// Mitsubishi GX Works2 project: 멜섹 485 통신 온도계   PLC: Q03UDV

PROGRAM MAIN
VAR
  u2k2k1 : BOOL;
  k2k1 : BOOL;
END_VAR
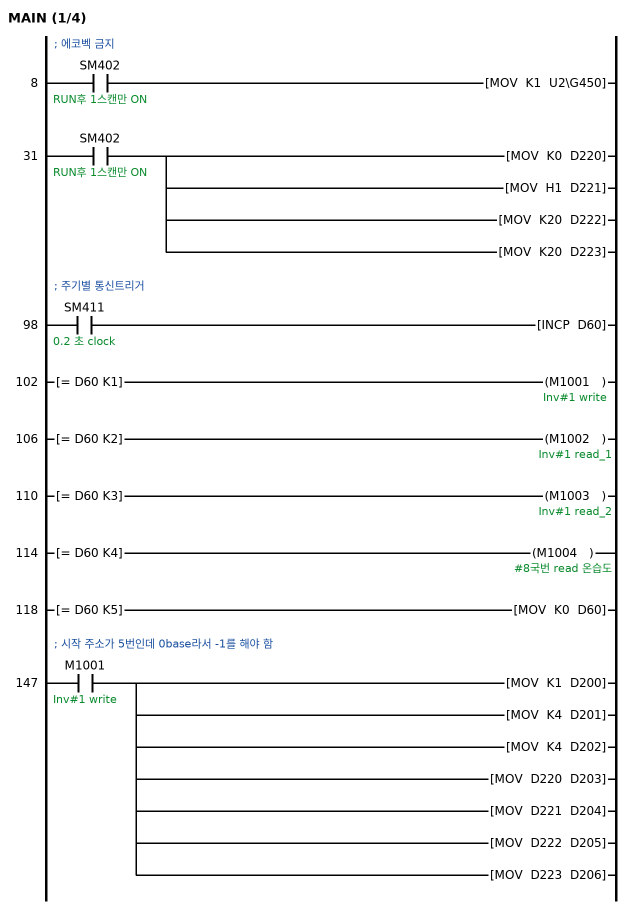
; 에코벡 금지
8     LD      SM402  ; RUN후 1스캔만 ON
      MOV     K1 U2\G450
        [note] 에코벡을 1로 만들어서 금지 시킴
31    LD      SM402  ; RUN후 1스캔만 ON
      MOV     K0 D220
        [note] 인버터 주파수 0hz설정
      MOV     H1 D221
        [note] 인버터 정지 값 1로만듬
      MOV     K20 D222
        [note] 가속 시간 초기값
      MOV     K20 D223
        [note] 감속 시간 초기값
; 주기별 통신트리거
98    LD      SM411  ; 0.2 초 clock
      INCP    D60
102   LD=     D60 K1
      OUT     M1001  ; Inv#1 write
106   LD=     D60 K2
      OUT     M1002  ; Inv#1 read_1
110   LD=     D60 K3
      OUT     M1003  ; Inv#1 read_2
114   LD=     D60 K4
      OUT     M1004  ; #8국번 read 온습도
118   LD=     D60 K5
      MOV     K0 D60
; 시작 주소가 5번인데 0base라서 -1를 해야 함
147   LD      M1001  ; Inv#1 write
      MOV     K1 D200
        [note] ; #1 WRITE DATA PLC>INV설정
      MOV     K4 D201
        [note] 5번인데 0base라서 -1를 한다
      MOV     K4 D202
      MOV     D220 D203
      MOV     D221 D204
      MOV     D222 D205
      MOV     D223 D206
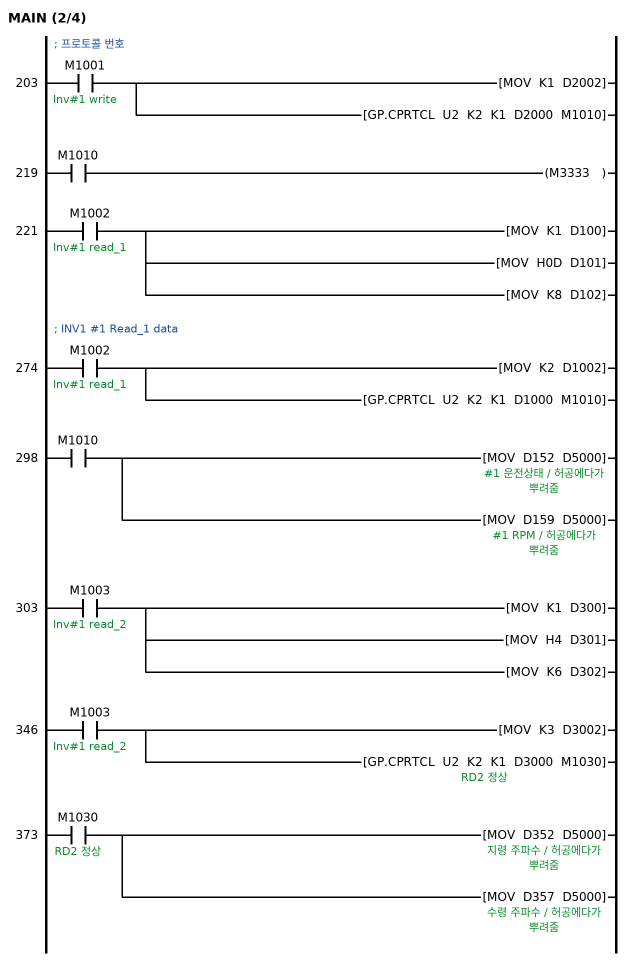
; 프로토콜 번호
203   LD      M1001  ; Inv#1 write
      MOV     K1 D2002
      GP.CPRTCL U2 K2 K1 D2000 M1010
219   LD      M1010
      OUT     M3333
221   LD      M1002  ; Inv#1 read_1
      MOV     K1 D100
        [note] SLAVE ADRESS #1
      MOV     H0D D101
        [note] START ADDRESS 000E-1=H0D
      MOV     K8 D102
        [note] 워드 주소개수
; INV1 #1 Read_1 data
274   LD      M1002  ; Inv#1 read_1
      MOV     K2 D1002
        [note] 프로토콜 2번
      GP.CPRTCL U2 K2 K1 D1000 M1010
298   LD      M1010
      MOV     D152 D5000  ; #1 운전상태 / 허공에다가 뿌려줌
      MOV     D159 D5000  ; #1 RPM
303   LD      M1003  ; Inv#1 read_2
      MOV     K1 D300
        [note] slave address #1
      MOV     H4 D301
        [note] start adress 5 -1
      MOV     K6 D302
        [note] 워드 주소갯수 6개 최대 8개
346   LD      M1003  ; Inv#1 read_2
      MOV     K3 D3002
        [note] 프로토콜 번호 3번
      GP.CPRTCL U2 K2 K1 D3000 M1030  ; RD2 정상
373   LD      M1030  ; RD2 정상
      MOV     D352 D5000  ; 지령 주파수
      MOV     D357 D5000  ; 수령 주파수
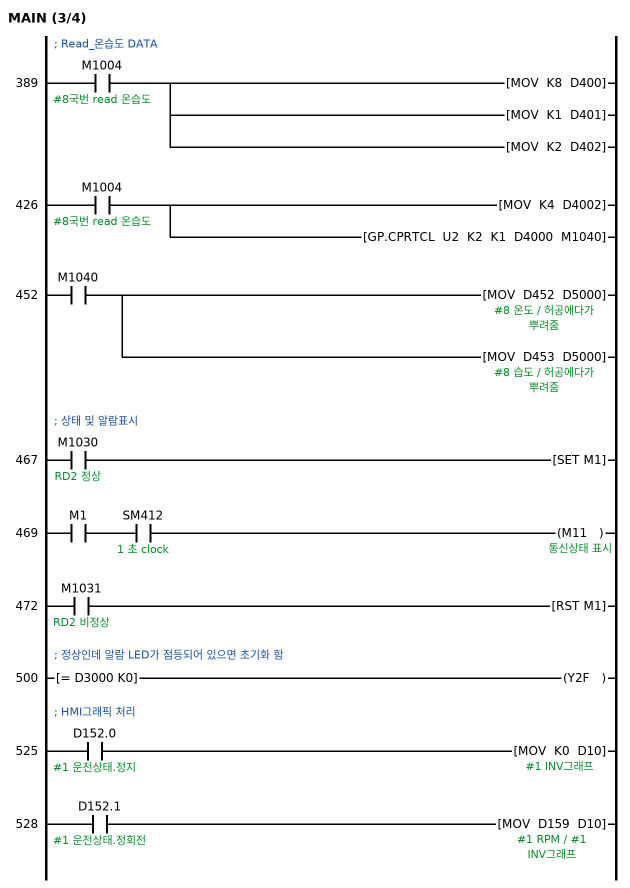
; Read_온습도 DATA
389   LD      M1004  ; #8국번 read 온습도
      MOV     K8 D400
        [note] #8 slave address
      MOV     K1 D401
        [note] start address 0001
      MOV     K2 D402
        [note] 워드 갯수 2개
426   LD      M1004  ; #8국번 read 온습도
      MOV     K4 D4002
        [note] 프로토콜 번호 4
      GP.CPRTCL U2 K2 K1 D4000 M1040
452   LD      M1040
      MOV     D452 D5000  ; #8 온도
      MOV     D453 D5000  ; #8 습도
; 상태 및 알람표시
467   LD      M1030  ; RD2 정상
      SET     M1
469   LD      M1
      AND     SM412  ; 1 초 clock
      OUT     M11  ; 통신상태 표시
472   LD      M1031  ; RD2 비정상
      RST     M1
; 정상인데 알람 LED가 점등되어 있으면 초기화 함
500   LD=     D3000 K0
      OUT     Y2F
        [note] 시리얼 알람 초기화
; HMI그래픽 처리
525   LD      D152.0  ; #1 운전상태.정지
      MOV     K0 D10  ; #1 INV그래프
528   LD      D152.1  ; #1 운전상태.정회전
      MOV     D159 D10
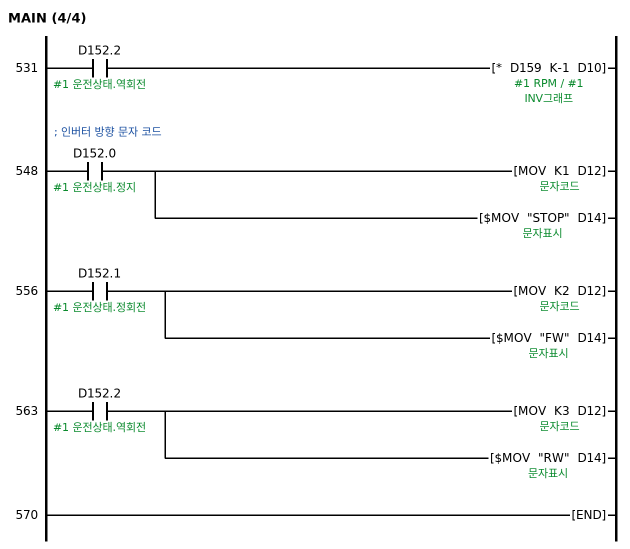
531   LD      D152.2  ; #1 운전상태.역회전
      *       D159 K-1 D10
; 인버터 방향 문자 코드
548   LD      D152.0  ; #1 운전상태.정지
      MOV     K1 D12  ; 문자코드
      $MOV    "STOP" D14  ; 문자표시
556   LD      D152.1  ; #1 운전상태.정회전
      MOV     K2 D12
      $MOV    "FW" D14
563   LD      D152.2  ; #1 운전상태.역회전
      MOV     K3 D12
      $MOV    "RW" D14
570   END
END_PROGRAM
